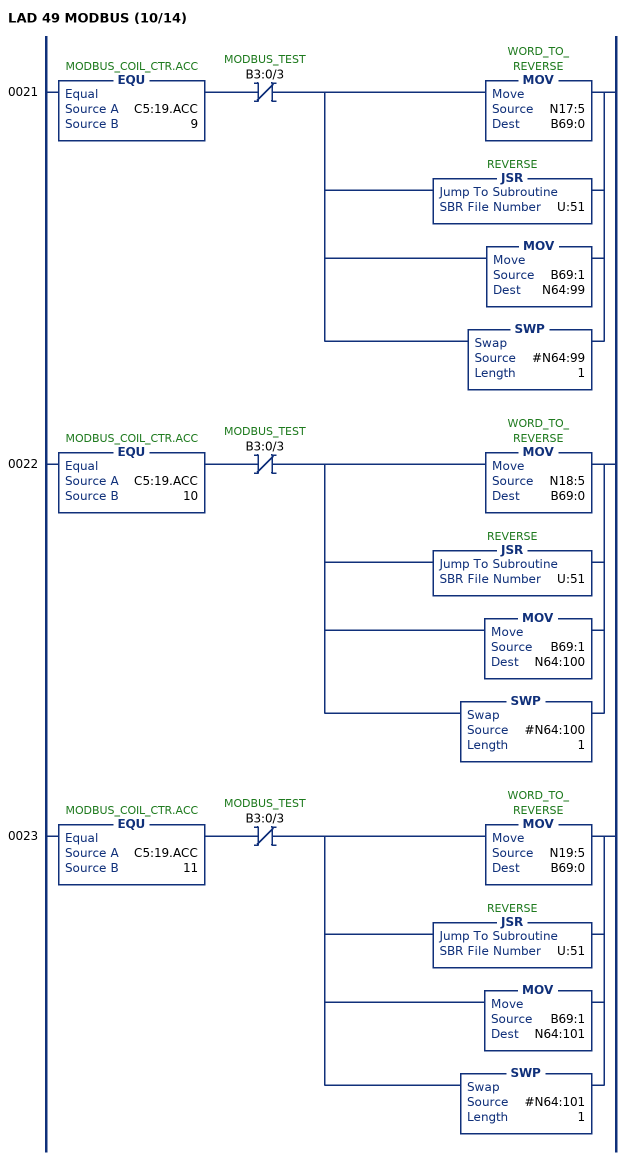
% Rung: 21 %
SOR EQU C5:19.ACC 9 XIO B3:0/3 BST MOV N17:5 B69:0 NXB JSR U:51 NXB MOV B69:1 N64:99 NXB SWP #N64:99 1 BND EOR
%   C5:19  MODBUS_COIL_CTR %
%   B3:0/3  MODBUS_TEST %
%   N17:5  ADS_B_ALARMS_0  "ALARM Alarm bits" %
%   B69:0  WORD_TO_REVERSE %
%   U:51  REVERSE %
%   B69:1  REVERSED_WORD %
% Rung: 22 %
SOR EQU C5:19.ACC 10 XIO B3:0/3 BST MOV N18:5 B69:0 NXB JSR U:51 NXB MOV B69:1 N64:100 NXB SWP #N64:100 1 BND EOR
%   C5:19  MODBUS_COIL_CTR %
%   B3:0/3  MODBUS_TEST %
%   N18:5  ADS_C_ALARMS_0 %
%   B69:0  WORD_TO_REVERSE %
%   U:51  REVERSE %
%   B69:1  REVERSED_WORD %
% Rung: 23 %
SOR EQU C5:19.ACC 11 XIO B3:0/3 BST MOV N19:5 B69:0 NXB JSR U:51 NXB MOV B69:1 N64:101 NXB SWP #N64:101 1 BND EOR
%   C5:19  MODBUS_COIL_CTR %
%   B3:0/3  MODBUS_TEST %
%   N19:5  ADS_D_ALARMS_0 %
%   B69:0  WORD_TO_REVERSE %
%   U:51  REVERSE %
%   B69:1  REVERSED_WORD %

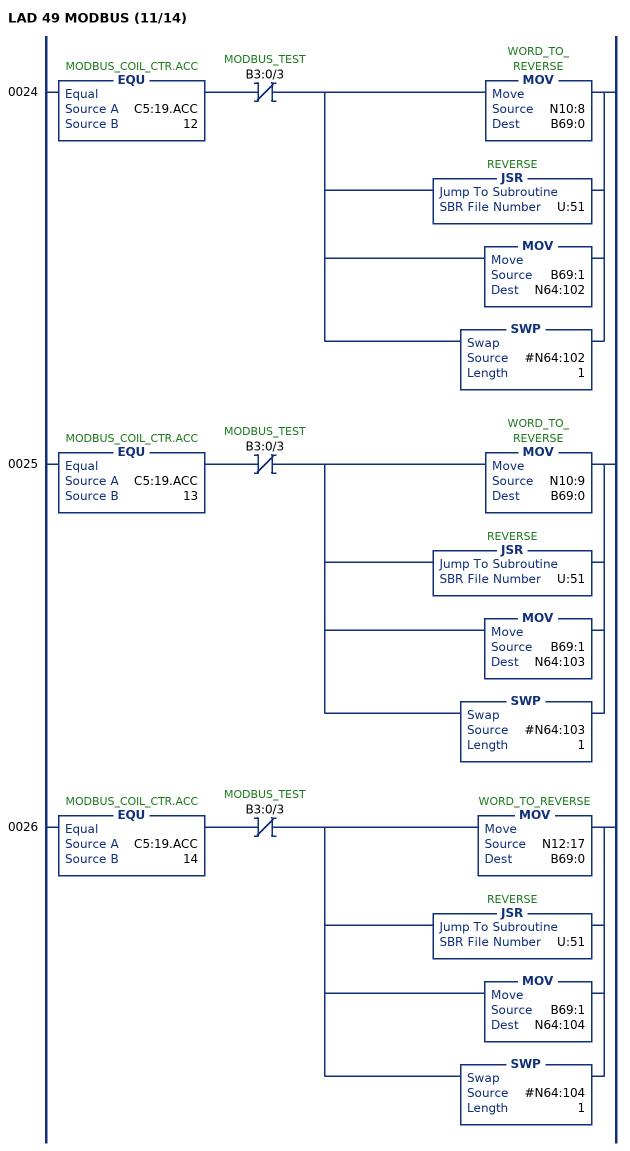
% Rung: 24 %
SOR EQU C5:19.ACC 12 XIO B3:0/3 BST MOV N10:8 B69:0 NXB JSR U:51 NXB MOV B69:1 N64:102 NXB SWP #N64:102 1 BND EOR
%   C5:19  MODBUS_COIL_CTR %
%   B3:0/3  MODBUS_TEST %
%   N10:8  SYSTEM_WARNINGS_0  "WARNING System Warnings" %
%   B69:0  WORD_TO_REVERSE %
%   U:51  REVERSE %
%   B69:1  REVERSED_WORD %
% Rung: 25 %
SOR EQU C5:19.ACC 13 XIO B3:0/3 BST MOV N10:9 B69:0 NXB JSR U:51 NXB MOV B69:1 N64:103 NXB SWP #N64:103 1 BND EOR
%   C5:19  MODBUS_COIL_CTR %
%   B3:0/3  MODBUS_TEST %
%   N10:9  SYSTEM_WARNINGS_1  "WARNING System Warnings" %
%   B69:0  WORD_TO_REVERSE %
%   U:51  REVERSE %
%   B69:1  REVERSED_WORD %
% Rung: 26 %
SOR EQU C5:19.ACC 14 XIO B3:0/3 BST MOV N12:17 B69:0 NXB JSR U:51 NXB MOV B69:1 N64:104 NXB SWP #N64:104 1 BND EOR
%   C5:19  MODBUS_COIL_CTR %
%   B3:0/3  MODBUS_TEST %
%   N12:17  PURIFY_WARNINGS_0 %
%   B69:0  WORD_TO_REVERSE %
%   U:51  REVERSE %
%   B69:1  REVERSED_WORD %

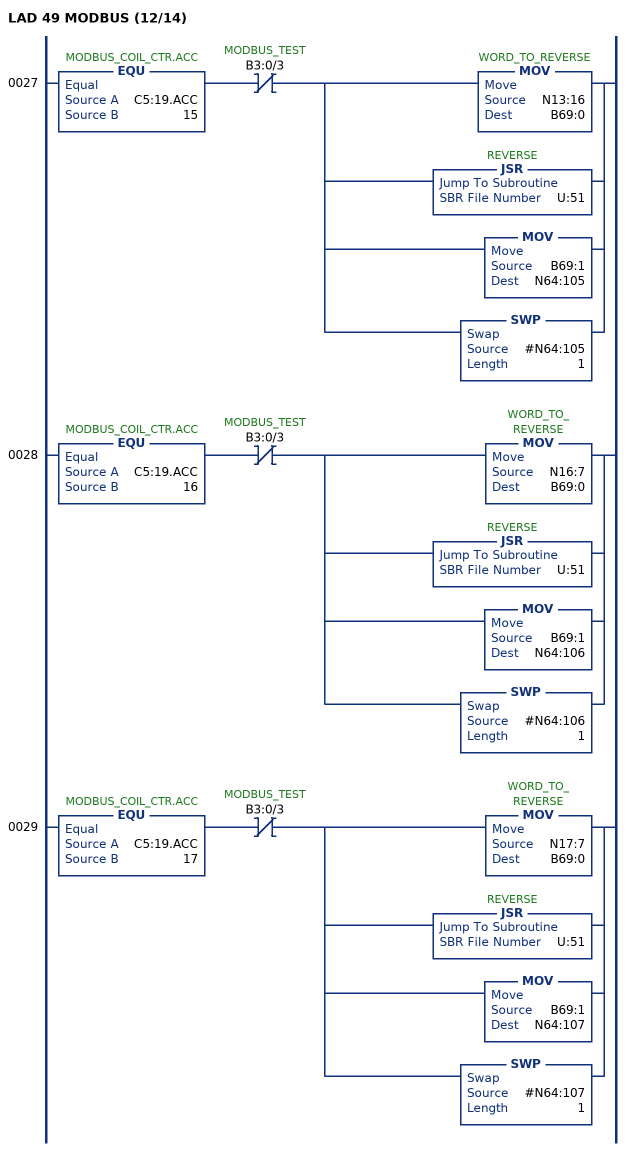
% Rung: 27 %
SOR EQU C5:19.ACC 15 XIO B3:0/3 BST MOV N13:16 B69:0 NXB JSR U:51 NXB MOV B69:1 N64:105 NXB SWP #N64:105 1 BND EOR
%   C5:19  MODBUS_COIL_CTR %
%   B3:0/3  MODBUS_TEST %
%   N13:16  REGEN_WARNINGS_0 %
%   B69:0  WORD_TO_REVERSE %
%   U:51  REVERSE %
%   B69:1  REVERSED_WORD %
% Rung: 28 %
SOR EQU C5:19.ACC 16 XIO B3:0/3 BST MOV N16:7 B69:0 NXB JSR U:51 NXB MOV B69:1 N64:106 NXB SWP #N64:106 1 BND EOR
%   C5:19  MODBUS_COIL_CTR %
%   B3:0/3  MODBUS_TEST %
%   N16:7  ADS_A_WARNINGS_0  "WARNING ADS A Warnings" %
%   B69:0  WORD_TO_REVERSE %
%   U:51  REVERSE %
%   B69:1  REVERSED_WORD %
% Rung: 29 %
SOR EQU C5:19.ACC 17 XIO B3:0/3 BST MOV N17:7 B69:0 NXB JSR U:51 NXB MOV B69:1 N64:107 NXB SWP #N64:107 1 BND EOR
%   C5:19  MODBUS_COIL_CTR %
%   B3:0/3  MODBUS_TEST %
%   N17:7  ADS_B_WARNINGS_0  "WARNING Warning bits" %
%   B69:0  WORD_TO_REVERSE %
%   U:51  REVERSE %
%   B69:1  REVERSED_WORD %

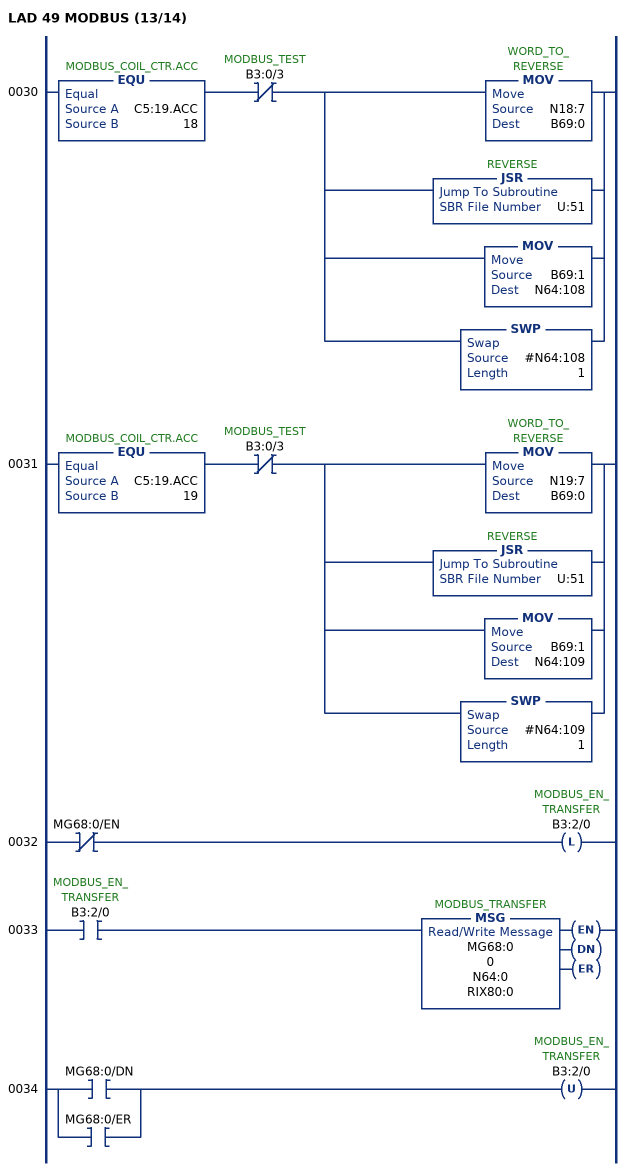
% Rung: 30 %
SOR EQU C5:19.ACC 18 XIO B3:0/3 BST MOV N18:7 B69:0 NXB JSR U:51 NXB MOV B69:1 N64:108 NXB SWP #N64:108 1 BND EOR
%   C5:19  MODBUS_COIL_CTR %
%   B3:0/3  MODBUS_TEST %
%   N18:7  ADS_C_WARNINGS_0 %
%   B69:0  WORD_TO_REVERSE %
%   U:51  REVERSE %
%   B69:1  REVERSED_WORD %
% Rung: 31 %
SOR EQU C5:19.ACC 19 XIO B3:0/3 BST MOV N19:7 B69:0 NXB JSR U:51 NXB MOV B69:1 N64:109 NXB SWP #N64:109 1 BND EOR
%   C5:19  MODBUS_COIL_CTR %
%   B3:0/3  MODBUS_TEST %
%   N19:7  ADS_D_WARNINGS_0 %
%   B69:0  WORD_TO_REVERSE %
%   U:51  REVERSE %
%   B69:1  REVERSED_WORD %
% Rung: 32 %
SOR XIO MG68:0/EN OTL B3:2/0 EOR
%   B3:2/0  MODBUS_EN_TRANSFER %
% Rung: 33 %
SOR XIC B3:2/0 MSG MG68:0 0 N64:0 RIX80:0 EOR
%   B3:2/0  MODBUS_EN_TRANSFER %
%   MSG set-up: CIP Generic | 33 | 0 | ? | 0 | 0 | 0 | 0 | 172.16.14.73 | 0 | 0 | 172.16.14.73 | RIX80:0 | 10 | 4 | 150 | 3 | 4 | 96 | 3 | 252 | N64:0 %
%   MG68:0  MODBUS_TRANSFER %
%   N64:0  REGISTER_START %
% Rung: 34 %
SOR BST XIC MG68:0/DN NXB XIC MG68:0/ER BND OTU B3:2/0 EOR
%   B3:2/0  MODBUS_EN_TRANSFER %

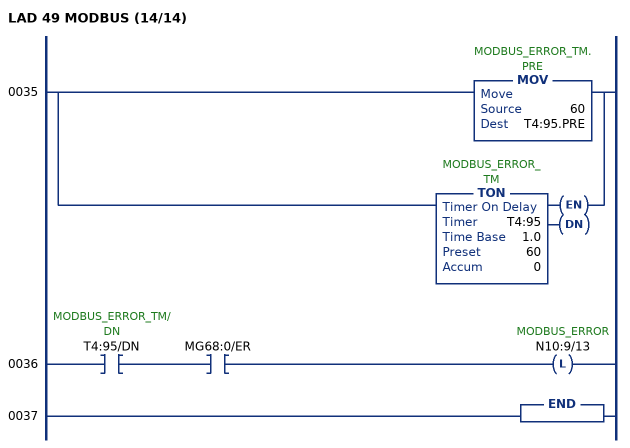
% Rung: 35 %
SOR BST MOV 60 T4:95.PRE NXB TON T4:95 1.0 60 0 BND EOR
%   T4:95  MODBUS_ERROR_TM %
% Rung: 36 %
SOR XIC T4:95/DN XIC MG68:0/ER OTL N10:9/13 EOR
%   T4:95  MODBUS_ERROR_TM %
%   N10:9/13  MODBUS_ERROR %
% Rung: 37 %
SOR END EOR

LADDER 50 "PLC_FAULT"
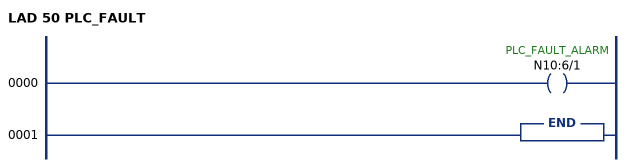
% Rung: 0 %
SOR OTE N10:6/1 EOR
%   N10:6/1  PLC_FAULT_ALARM %
% Rung: 1 %
SOR END EOR

LADDER 51 "REVERSE"
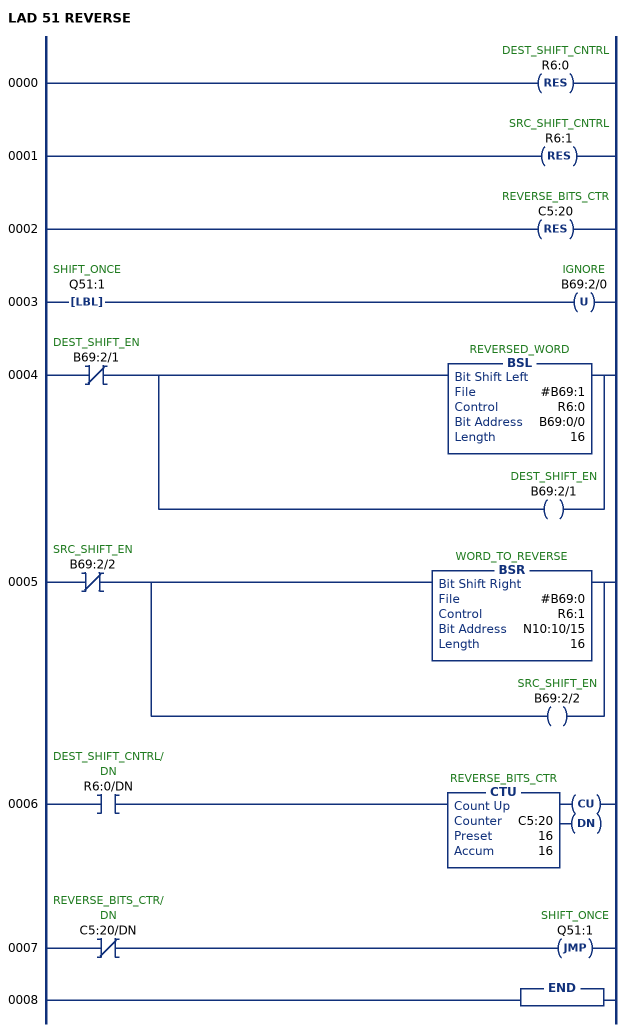
% Rung: 0 %
SOR RES R6:0 EOR
%   R6:0  DEST_SHIFT_CNTRL %
% Rung: 1 %
SOR RES R6:1 EOR
%   R6:1  SRC_SHIFT_CNTRL %
% Rung: 2 %
SOR RES C5:20 EOR
%   C5:20  REVERSE_BITS_CTR %
% Rung: 3 %
SOR LBL Q51:1 OTU B69:2/0 EOR
%   Q51:1  SHIFT_ONCE %
%   B69:2/0  IGNORE %
% Rung: 4 %
SOR XIO B69:2/1 BST BSL #B69:1 R6:0 B69:0/0 16 NXB OTE B69:2/1 BND EOR
%   B69:2/1  DEST_SHIFT_EN %
%   B69:1  REVERSED_WORD %
%   R6:0  DEST_SHIFT_CNTRL %
% Rung: 5 %
SOR XIO B69:2/2 BST BSR #B69:0 R6:1 N10:10/15 16 NXB OTE B69:2/2 BND EOR
%   B69:2/2  SRC_SHIFT_EN %
%   B69:0  WORD_TO_REVERSE %
%   R6:1  SRC_SHIFT_CNTRL %
%   N10:10/15  ALWAYS_OFF  "If this is off, go ahead and turn it off" %
% Rung: 6 %
SOR XIC R6:0/DN CTU C5:20 16 16 EOR
%   R6:0  DEST_SHIFT_CNTRL %
%   C5:20  REVERSE_BITS_CTR %
% Rung: 7 %
SOR XIO C5:20/DN JMP Q51:1 EOR
%   C5:20  REVERSE_BITS_CTR %
%   Q51:1  SHIFT_ONCE %
% Rung: 8 %
SOR END EOR

OTHER DOCUMENTED ADDRESSES
  B30:0  CONFIG_BITS_HARDWARE  "CONFIG Hardware options installed"
  B30:5  SYSTEM_STATUS_0  "STATUS System Status of system contro entities"
  B31:2  SYSTEM_HMI_CMD_0  "COMMAND HMI Commands"
  B31:3  SYSTEM_HMI_CMD_1  "COMMAND HMI Commands"
  B31:4  SYSTEM_HMI_CMD_2  "COMMAND HMI Commands"
  B31:5  SYSTEM_HMI_CMD_3
  B31:6  SYSTEM_HMI_CMD_4  "COMMAND HMI Commands"
  B31:7  SYSTEM_HMI_CMD_5  "COMMAND HMI Commands"
  B33:0  PURIFY_HMI_CMDS
  B33:0/1  DEF_PURIFY_MAX  "COMMAND HMI Purifier Max Time Load Defaults"
  B34:0  REGEN_HMI_CMDS
  B34:2  REGEN_FLAGS
  B35:2  MANUAL_HMI_CMNDS_0
  DFILE:0  "OUTPUT"
  DFILE:1  "INPUT"
  DFILE:2  "STATUS"
  DFILE:3  "BINARY"
  DFILE:4  "TIMER"
  DFILE:5  "COUNTER"
  DFILE:6  "CONTROL"
  DFILE:7  "SYSTEM CFG Maintains the values that characterize t he system"
  DFILE:8  "FLOAT"
  DFILE:9  "CONSTANTS The collection of sy stem and subsystem c onstants"
  DFILE:10  "SYSTEM Contain the values f or system control"
  DFILE:11  "PROCESS Contains the values for the processing m achine"
  DFILE:12  "PURIFY Contains the values required for purify"
  DFILE:13  "REGEN Contains the values required for regen"
  DFILE:14  "BYPASS"
  DFILE:15  "MANUAL CTL Contains the data fo r the manual valve c ontrol"
  DFILE:16  "ADSORBER_A Contains the values for Adsorber A"
  DFILE:17  "ADSORBER_B Contains the values required for Adsorbe r B"
  DFILE:18  "ADSORBER_C"
  DFILE:19  "ADSORBER_D"
  DFILE:20  "MIX PANEL"
  DFILE:21  "OUTLET"
  DFILE:23  "MB_HRTBT"
  DFILE:25  "PID HEATER"
  DFILE:30  "SYSTEM CFG"
  DFILE:31  "SYSTEM"
  DFILE:32  "PROCESS"
  DFILE:33  "PURIFY"
  DFILE:34  "REGEN"
  DFILE:35  "MANUAL CTL"
  DFILE:38  "HEATERS"
  DFILE:51  "TOTAL_FLOW"
  DFILE:52  "SERIAL"
  DFILE:64  "MODBUS"
  DFILE:68  "TRANSFER"
  DFILE:69  "REVERSE"
  DFILE:80  "MSG_SETUP"
  N7:0  CONFIG_BITS_ALM
  N7:1  CONFIG_BITS_ALM_O  "CONFIG System alarms enable"
  N7:2  CONFIG_BITS_ALM_1  "CONFIG System alarms enable"
  N7:3  CONFIG_BITS_WARN_0  "CONFIG System warnings enable"
  N7:4  CONFIG_BITS_WARN_1  "CONFIG System warnings enable"
  N7:5  CONFIG_BITS_WARN
  N7:6  CONFIG_OPEN_TC_ALM
  N7:7  CONFIG_OPEN_TC_WARN
  N10:10  SYSTEM_CONTROL  "CONTROL System Bits used to manipulate hardware"
  N10:16  SYSTEM_FLAGS_1
  N12:4  PURIFY_FLAGS_0  "STATUS Flags used by the purify process"
  N12:5  PURIFY_CONTROL  "CONTROL Control bits used by the purify process to change hardware states"
  N12:12  PURIFY_CALC_0  "CONFIG Math result placeholder for the purify time calculation"
  N12:13  PURIFY_FACTOR_TIME  "CONFIG The factored purify time accounting for the purify percent factor (hours)"
  N12:14  PURIFY_MAX_TIME
  N13:5  REGEN_CONTROL  "CONTROL Regen Bits used to manipulate hardware"
  N14:1  BYPASS_COMMAND
  N15:4  MANUAL_FLAGS_0
  N16:3  ADS_A_FLAGS_0  "STATUS Flags used for Adsorber A"
  N17:3  ADS_B_FLAGS_0  "STATUS Flags used for Adsorber B"
  PD25:0.5  "PID ADS Preheater Derivative Term"
  PD25:0.13  "PID ADS Preheater Loop Update Time"
  PD25:1.5  "PID ADS A Blanket Derivative Term"
  PD25:1.13  "PID ADS A Blanket Loop Update Time"
  PD25:3.5  "PID ADS B Blanket Derivative Term"
  PD25:3.13  "PID ADS B Blanket Loop Update Time"
  PD25:4.5  "PID ADS C Blanket Derivative Term"
  PD25:4.13  "PID ADS C Blanket Loop Update Time"
  PD25:5.5  "PID ADS D Blanket Derivative Term"
  PD25:5.13  "PID ADS D Blanket Loop Update Time"

COMMENTS NOT ATTACHED TO A CURRENT RUNG
  N10:26: MFM / CONFIGURE MFM AND FLOW
  N13:14/12: ADS A Gas Temp Thermocouple alarm
    If the alarm conditions are met, latch the alarm.
    If the operator acknowledges, reset it.
  U:29: Call the routine to operate the Adsorber D fault control
  N7:8: Scale analog inputs / TODO: Do we need to add the ability to adjust the ammonia sensor scaling?
  N16:5/1: OPEN TC's
  N18:5/7: If the delay timer has completed, latch the alarm.
    If the operator acknowledges, reset it.
  T4:81: UPS Failed Warning

REVISION NOTES
  0: moved some bits out of N7 into B30
  1: moved bits out of N10 into B31
  2: moved bits from N15 into B35
  3: added the final data files. didn't need to move any bits
  4: updated configuration for TC and AI cards. updated DO module point assignments
  5: added logic for double-acting purify valves
  6: added rod and blanket limits
  7: added tags for default buttons
  8: cleaning up bed b pid control code
  9: removed h2 sensor and moved moisture sensor to channel 6
  10: changed processor name
  11: added px3 reading
  12: added call to mix panel routine
  13: test ok
  14: trying to clear plc fault by entering new pid default parameters
  15: changed stored PID values so that it maybe doesn't fault the PLC
  16: copid in new PID values from PS21
  17: cleared out the data table
  18: changed ADS_TC_OPEN_SP to 13700 by default
  19: setting default PID parameters
  20: added in preheater and blanket setpoints
  21: lots of changes to PID control
  22: fixed up PID defaults
  23: done testing
  24: got rid of separate PID defaults
  25: fixed loop update time bug in preheater defaults
  26: PID control done
  27: ok, now it's done. made Adsorber B use the same PID parameters as Adsorber A.
  28: added control for AV11 to system routine
  29: moved mixing panel valves into mixing panel routine
  30: some small fixes to the processing subroutine.
  31: cleaned up manual valve control for AV10, 11
  32: minor edit to purify factor calculation
  33: made some fixes to ADS_A routine including adding another state buffer for adsorber-only alarms.
  34: fixed up ADS_B routine so that it's like ADS_B
  35: Regen sequence modified and default regen paramters added
  36: added regen default comments
  37: added regen steps to constants
  38: Regen counter condition resets added
  39: Fixed regen standby buffer
  40: Regen buffering and sequencing checked and fixed
  41: Merged
  42: remove alarm aknowledge
  43: Updated alarm tag names
  44: PH fault changed
  45: manual mode PID taop PID control
  46: Added fail to cool alarm and warning
  47: trying to fix ph fault
  48: fixing open tc
  49: fixed open tc logic
  50: ok, now it's fixed

DATA TABLE (non-zero values as saved)
DATA T4
% .PRE .ACC %
% T4:0 % 2 0
% T4:1 % 60 18
% T4:2 % 2 0
% T4:3 % 2 0
% T4:4 % 60 0
% T4:5 % 60 0
% T4:6 % 1000 111
% T4:7 % 1000 111
% T4:8 % 5 0
% T4:9 % 5 0
% T4:10 % 5 0
% T4:11 % 5 0
% T4:12 % 5 0
% T4:13 % 5 0
% T4:14 % 5 0
% T4:15 % 5 0
% T4:16 % 21600 0
% T4:17 % 21600 0
% T4:18 % 60 0
% T4:19 % 21600 0
% T4:20 % 5 0
% T4:21 % 5 0
% T4:22 % 5 0
% T4:23 % 5 0
% T4:24 % 1 0
% T4:25 % 1 0
% T4:26 % 30 0
% T4:27 % 30 0
% T4:28 % 5 0
% T4:29 % 5 0
% T4:30 % 60 0
% T4:31 % 60 0
% T4:32 % 5 0
% T4:33 % 5 0
% T4:34 % 5 0
% T4:35 % 5 0
% T4:36 % 5 0
% T4:37 % 5 0
% T4:38 % 10 0
% T4:39 % 60 0
% T4:40 % 5 0
% T4:41 % 5 0
% T4:42 % 5 0
% T4:43 % 5 0
% T4:44 % 5 0
% T4:45 % 5 0
% T4:46 % 5 0
% T4:47 % 5 0
% T4:48 % 5 0
% T4:49 % 5 0
% T4:50 % 5 0
% T4:51 % 5 0
% T4:52 % 2 0
% T4:53 % 2 0
% T4:54 % 500 77
% T4:55 % 60 0
% T4:56 % 60 0
% T4:57 % 30 0
% T4:58 % 30 30
% T4:59 % 60 0
% T4:60 % 60 0
% T4:61 % 10 0
% T4:62 % 10 0
% T4:63 % 60 0
% T4:64 % 60 0
% T4:65 % 60 0
% T4:66 % 60 0
% T4:67 % 60 0
% T4:68 % 60 0
% T4:69 % 60 0
% T4:70 % 5 0
% T4:71 % 5 0
% T4:72 % 5 0
% T4:73 % 5 0
% T4:74 % 60 0
% T4:75 % 60 0
% T4:76 % 5 0
% T4:77 % 5 0
% T4:78 % 10 0
% T4:79 % 10 0
% T4:80 % 5 0
% T4:81 % 5 0
% T4:82 % 5 0
% T4:83 % 5 0
% T4:84 % 5 0
% T4:85 % 5 0
% T4:86 % 5 0
% T4:87 % 5 0
% T4:88 % 5 0
% T4:89 % 5 0
% T4:90 % 21600 0
% T4:91 % 21600 0
% T4:92 % 21600 0
% T4:93 % 21600 61
% T4:94 % 5 5
% T4:95 % 60 0
% T4:96 % 500 0
% T4:97 % 5 0
% T4:98 % 5 0
% T4:99 % 1 0
% T4:100 % 180 0
% T4:101 % 60 0
% T4:119 % 120 0
% T4:120 % 60 0
% T4:121 % 60 0
% T4:122 % 5 0
% T4:123 % 5 0
% T4:124 % 5 0
% T4:126 % 5 0
% T4:127 % 5 5
% T4:128 % 5 0
% T4:129 % 5 5
% T4:130 % 5 0
% T4:131 % 5 0
% T4:132 % 5 0
% T4:133 % 5 0
% T4:134 % 5 0
% T4:136 % 5 0
% T4:138 % 5 0
% T4:140 % 5 0
DATA C5
% .PRE .ACC %
% C5:0 % 48 1
% C5:1 % 60 40
% C5:2 % 24 20
% C5:3 % 32767 2
% C5:4 % 240 0
% C5:5 % 180 0
% C5:7 % 10 0
% C5:8 % 480 0
% C5:9 % 5 0
% C5:10 % 5 0
% C5:11 % 5 0
% C5:12 % 5 0
% C5:13 % 30 0
% C5:14 % 10 0
% C5:17 % 720 0
% C5:18 % 720 0
% C5:19 % 20 11
% C5:20 % 16 16
% C5:21 % 30 0
DATA R6
% .LEN .POS %
% R6:0 % 16 0
% R6:1 % 16 0
DATA T23
% .PRE .ACC %
% T23:1 % 100 0
% T23:2 % 100 0
